// TIA Portal V15.1 export
// export: Created 2024-06-21T08:41:11.5404395Z, ExportSetting WithDefaults, DisplayName Totally Integrated Automation Portal, DisplayVersion V15.1 Update 5, DisplayName TIA Portal Openness, DisplayVersion V15.1 Update 5, DisplayName SINAMICS Startdrive Advanced, DisplayVersion V15.1, DisplayName G130, G150, S120, S150, SINAMICS MV, S210, DisplayVersion V15.1, DisplayName G110M, G120, G120C, G120D, G120P, DisplayVersion V15.1, DisplayName STEP 7 Professional, DisplayVersion V15.1 Update 5, DisplayName STEP 7 Safety, DisplayVersion V15.1, DisplayName WinCC Professional, DisplayVersion V15.1 Update 5, DisplayName SIMATIC Visualization Architect, DisplayVersion V15.1
FUNCTION "LGBShiftRegLine-Config" : Void   // FC6644, FBD
TITLE = LMovUnit2Pos1S-C-Config / LGBShiftRegLine-Config
{ S7_Optimized_Access := 'FALSE' }
AUTHOR : VCC
FAMILY : Control
NAME : Bit2Word
VERSION : 1.0
// =============================================================================
// Move Configuration
// =============================================================================
// stored: AutoNumber false, IsIECCheckEnabled false, SetENOAutomatically False, UDAEnableTagReadback false
   VAR_INPUT
      C_BodyPitch : Int;   // Setpoint Body pitch (cm)
      C_CycleTime : Int;   // Setpoint Cycle time (sec)
      C_NbrOfWorkZones : Int;   // Number of work zones (Andon positions)
      C_TriggerDetPosition : DInt;   // Position trigger sensor
      C_InfeedConvStopDetPosition : DInt;   // Position stop sensor of infeed conveyor (usually negative)
      C_EncPlsCntrMin : DInt;   // Encoder pulse counter - minimum value
      C_EncPlsCntrMax : DInt;   // Encoder pulse counter - maximum value
      "C_Sealing/Paint/PreTreatment" : Int;   // Pop-up choise -> 1 = Sealing ; 2 = Paint ; 3 = PreTreatment
      C_Area1_Used : Bool;   // AREA is used
      C_Area1_InZoneX : Int;   // In which zone the AREA is located
      C_Area1_StartPosition : Int;   // Start position (cm) for the AREA in that zone
      C_Area1_EndPosition : Int;   // Stop position (cm) for the AREA in that zone
      C_Area2_Used : Bool;   // AREA is used
      C_Area2_InZoneX : Int;   // In which zone the AREA is located
      C_Area2_StartPosition : Int;   // Start position (cm) for the AREA in that zone
      C_Area2_EndPosition : Int;   // Stop position (cm) for the AREA in that zone
      C_Area3_Used : Bool;   // AREA is used
      C_Area3_InZoneX : Int;   // In which zone the AREA is located
      C_Area3_StartPosition : Int;   // Start position (cm) for the AREA in that zone
      C_Area3_EndPosition : Int;   // Stop position (cm) for the AREA in that zone
      C_Area4_Used : Bool;   // AREA is used
      C_Area4_InZoneX : Int;   // In which zone the AREA is located
      C_Area4_StartPosition : Int;   // Start position (cm) for the AREA in that zone
      C_Area4_EndPosition : Int;   // Stop position (cm) for the AREA in that zone
      C_Area5_Used : Bool;   // AREA is used
      C_Area5_InZoneX : Int;   // In which zone the AREA is located
      C_Area5_StartPosition : Int;   // Start position (cm) for the AREA in that zone
      C_Area5_EndPosition : Int;   // Stop position (cm) for the AREA in that zone
      C_Area6_Used : Bool;   // AREA is used
      C_Area6_InZoneX : Int;   // In which zone the AREA is located
      C_Area6_StartPosition : Int;   // Start position (cm) for the AREA in that zone
      C_Area6_EndPosition : Int;   // Stop position (cm) for the AREA in that zone
      C_Area7_Used : Bool;   // AREA is used
      C_Area7_InZoneX : Int;   // In which zone the AREA is located
      C_Area7_StartPosition : Int;   // Start position (cm) for the AREA in that zone
      C_Area7_EndPosition : Int;   // Stop position (cm) for the AREA in that zone
      C_Area8_Used : Bool;   // AREA is used
      C_Area8_InZoneX : Int;   // In which zone the AREA is located
      C_Area8_StartPosition : Int;   // Start position (cm) for the AREA in that zone
      C_Area8_EndPosition : Int;   // Stop position (cm) for the AREA in that zone
      C_Area9_Used : Bool;   // AREA is used
      C_Area9_InZoneX : Int;   // In which zone the AREA is located
      C_Area9_StartPosition : Int;   // Start position (cm) for the AREA in that zone
      C_Area9_EndPosition : Int;   // Stop position (cm) for the AREA in that zone
      C_Area10_Used : Bool;   // AREA is used
      C_Area10_InZoneX : Int;   // In which zone the AREA is located
      C_Area10_StartPosition : Int;   // Start position (cm) for the AREA in that zone
      C_Area10_EndPosition : Int;   // Stop position (cm) for the AREA in that zone
   END_VAR
   VAR_IN_OUT
      IO_Config : "ShiftRegLineConfig";   // Output Word / Config
   END_VAR
BEGIN

REGION Network 1: **** 1 - Inputs **** Move Config
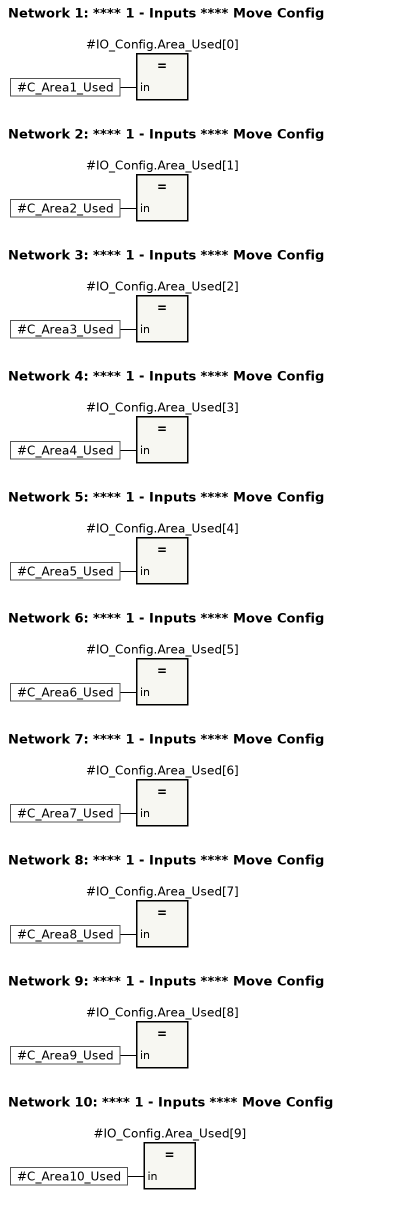
   #IO_Config.Area_Used[0] := #C_Area1_Used;
END_REGION

REGION Network 2: **** 1 - Inputs **** Move Config
   #IO_Config.Area_Used[1] := #C_Area2_Used;
END_REGION

REGION Network 3: **** 1 - Inputs **** Move Config
   #IO_Config.Area_Used[2] := #C_Area3_Used;
END_REGION

REGION Network 4: **** 1 - Inputs **** Move Config
   #IO_Config.Area_Used[3] := #C_Area4_Used;
END_REGION

REGION Network 5: **** 1 - Inputs **** Move Config
   #IO_Config.Area_Used[4] := #C_Area5_Used;
END_REGION

REGION Network 6: **** 1 - Inputs **** Move Config
   #IO_Config.Area_Used[5] := #C_Area6_Used;
END_REGION

REGION Network 7: **** 1 - Inputs **** Move Config
   #IO_Config.Area_Used[6] := #C_Area7_Used;
END_REGION

REGION Network 8: **** 1 - Inputs **** Move Config
   #IO_Config.Area_Used[7] := #C_Area8_Used;
END_REGION

REGION Network 9: **** 1 - Inputs **** Move Config
   #IO_Config.Area_Used[8] := #C_Area9_Used;
END_REGION

REGION Network 10: **** 1 - Inputs **** Move Config
   #IO_Config.Area_Used[9] := #C_Area10_Used;
END_REGION

NETWORK
TITLE = **** 1 Inputs **** Move Config UDT
// Move Config
      L     #C_BodyPitch;
      T     #IO_Config.BodyPitch;
      L     #C_CycleTime;
      T     #IO_Config.CycleTime;
      L     #C_NbrOfWorkZones;
      T     #IO_Config.NbrOfWorkZones;

      L     #C_InfeedConvStopDetPosition;
      T     #IO_Config.InfeedConvStopDetPosition;
      L     #C_TriggerDetPosition;
      T     #IO_Config.TriggerDetPosition;
      L     #C_EncPlsCntrMin;
      T     #IO_Config.EncPlsCntrMin;
      L     #C_EncPlsCntrMax;
      T     #IO_Config.EncPlsCntrMax;

      L     #"C_Sealing/Paint/PreTreatment";
      T     #IO_Config."Sealing/Paint/PreTreatment";

      L     #C_Area1_InZoneX;
      T     #IO_Config.Area_InZoneX[0];
      L     #C_Area1_StartPosition;
      T     #IO_Config.Area_StartPosition[0];
      L     #C_Area1_EndPosition;
      T     #IO_Config.Area_EndPosition[0];

      L     #C_Area2_InZoneX;
      T     #IO_Config.Area_InZoneX[1];
      L     #C_Area2_StartPosition;
      T     #IO_Config.Area_StartPosition[1];
      L     #C_Area2_EndPosition;
      T     #IO_Config.Area_EndPosition[1];

      L     #C_Area3_InZoneX;
      T     #IO_Config.Area_InZoneX[2];
      L     #C_Area3_StartPosition;
      T     #IO_Config.Area_StartPosition[2];
      L     #C_Area3_EndPosition;
      T     #IO_Config.Area_EndPosition[2];

      L     #C_Area4_InZoneX;
      T     #IO_Config.Area_InZoneX[3];
      L     #C_Area4_StartPosition;
      T     #IO_Config.Area_StartPosition[3];
      L     #C_Area4_EndPosition;
      T     #IO_Config.Area_EndPosition[3];

      L     #C_Area5_InZoneX;
      T     #IO_Config.Area_InZoneX[4];
      L     #C_Area5_StartPosition;
      T     #IO_Config.Area_StartPosition[4];
      L     #C_Area5_EndPosition;
      T     #IO_Config.Area_EndPosition[4];

      L     #C_Area6_InZoneX;
      T     #IO_Config.Area_InZoneX[5];
      L     #C_Area6_StartPosition;
      T     #IO_Config.Area_StartPosition[5];
      L     #C_Area6_EndPosition;
      T     #IO_Config.Area_EndPosition[5];

      L     #C_Area7_InZoneX;
      T     #IO_Config.Area_InZoneX[6];
      L     #C_Area7_StartPosition;
      T     #IO_Config.Area_StartPosition[6];
      L     #C_Area7_EndPosition;
      T     #IO_Config.Area_EndPosition[6];

      L     #C_Area8_InZoneX;
      T     #IO_Config.Area_InZoneX[7];
      L     #C_Area8_StartPosition;
      T     #IO_Config.Area_StartPosition[7];
      L     #C_Area8_EndPosition;
      T     #IO_Config.Area_EndPosition[7];

      L     #C_Area9_InZoneX;
      T     #IO_Config.Area_InZoneX[8];
      L     #C_Area9_StartPosition;
      T     #IO_Config.Area_StartPosition[8];
      L     #C_Area9_EndPosition;
      T     #IO_Config.Area_EndPosition[8];

      L     #C_Area10_InZoneX;
      T     #IO_Config.Area_InZoneX[9];
      L     #C_Area10_StartPosition;
      T     #IO_Config.Area_StartPosition[9];
      L     #C_Area10_EndPosition;
      T     #IO_Config.Area_EndPosition[9];
END_FUNCTION
